// FBs/CSV/FB_EscreveCSVPonteiro
FUNCTION_BLOCK FB_EscreveCSVPonteiro
VAR_INPUT
	bInicia : BOOL;
	sNetId			: T_AmsNetId;	(* TwinCAT system network address *)
	sFileName	: T_MaxString;(* CSV destination file path and name *)
	MAX_CSV_COLUMNS : UINT;
	MAX_CSV_ROWS	: UINT;
	ppDataBase : POINTER TO POINTER TO STRING(255);
END_VAR
VAR_IN_OUT
	//database : ARRAY[*,*] OF STRING(255);
END_VAR
VAR_OUTPUT
	bBusy			: BOOL;
	bError			: BOOL;
	nErrId			: UDINT;
	nRow	 		: UDINT 	:= 0;(* Row number (record) *)
END_VAR
VAR
	bWrite			: BOOL := FALSE;(* Rising edge starts program execution *)
	sCSVLine		: T_MaxString := '';(* Single CSV text line (row, record), we are using string as record buffer (your are able to see created fields) *)
	sCSVField		: T_MaxString := '';(* Single CSV field value (column, record field) *)
	nColumn		: UDINT 	:= 0;(* Column number (record field) *)
	hFile			: UINT		:= 0;(* File handle of the source file *)
	step			: DWORD 	:= 0;
	fbFileOpen	: FB_FileOpen;(* Opens file *)
	fbFileClose	: FB_FileClose;(* Closes file *)
	fbFilePuts		: FB_FilePuts;(* Writes one record (line) *)
	fbWriter		: FB_CSVMemBufferWriter;(* Helper function block used to create CSV data bytes (single record line) *)
	rtInicia		: R_TRIG;
	

	MAX_CSV_FIELD_LENGTH : UDINT := 255;
END_VAR

IF xLicensaValida87208720 THEN
	
//Criado por Tiago Bortolini Cunico
	
	
	CASE step OF
		0:	(* Wait for rising edge at bWrite variable *)
			rtInicia(CLK:=bInicia , Q=> );//gera borda de subina quando liga	
			IF rtInicia.q THEN
				bWrite := TRUE;
			END_IF
			
			IF bWrite THEN
				bWrite 		:= FALSE;
				bBusy 		:= TRUE;
				bError		:= FALSE;
				nErrId		:= 0;
				hFile		:= 0;
				nRow	 	:= 0;
				nColumn		:= 0;
				step 		:= 1;
			END_IF
	
		1:	(* Open source file *)
			fbFileOpen(  bExecute := FALSE  );
			fbFileOpen( 	sNetId := sNetId, sPathName := sFileName, nMode := FOPEN_MODEAPPEND OR FOPEN_MODETEXT,(* Open file in TEXT mode!   FOPEN_MODEWRITE OR FOPEN_MODETEXT*)
							ePath := PATH_GENERIC, bExecute := TRUE );
			step := 2;
	
		2:(* Wait until open not busy *)
			fbFileOpen( bExecute := FALSE, bError => bError, nErrID => nErrID, hFile => hFile );
			IF NOT fbFileOpen.bBusy THEN
				IF NOT fbFileOpen.bError THEN
					step := 3;
				ELSE(* Error: file not found? *)
					step := 100;
				END_IF
			END_IF
	
		3:(* Convert one PLC record to CSV format *)
			sCSVLine := '';
			fbWriter.eCmd := eEnumCmd_First;(* Write first field value *)
			IF nRow < MAX_CSV_ROWS THEN
	
				FOR nColumn := 0 TO MAX_CSV_COLUMNS - 1 BY 1 DO	
					IF  ppDataBase <> 0 AND ppDataBase[nColumn] <> 0 THEN
						IF ppDataBase[nColumn][nRow] <>  '' THEN 
				
							sCSVField := STRING_TO_CSVFIELD( ppDataBase[nColumn][nRow], TRUE );(* TODO: Get field value from your application *)//sCSVField := STRING_TO_CSVFIELD( database[ nRow, nColumn ], FALSE );(* TODO: Get field value from your application *)
							
							(* Add new field to the record buffer *)
							fbWriter( 	pBuffer := ADR( sCSVLine ), cbBuffer := SIZEOF( sCSVLine ) - 1, putValue := sCSVField, pValue := 0, cbValue := 0,
										bCRLF := ( nColumn = MAX_CSV_COLUMNS-1 ) );(* bCRLF == TRUE => Write CRLF after the last field value *)
							IF fbWriter.bOk THEN
								fbWriter.eCmd := eEnumCmd_Next;(* Write next field value *)
							ELSE(* Error *)
								step := 100;
								RETURN;
							END_IF
						END_IF
					ELSE
						step := 100;
					END_IF
				END_FOR(* FOR nColumn := 0... *)
	
				(* FB_FilePuts adds allready CR (carriage return) to the written line.
				We have to replace the $R$L characters with $L character to avoid double CR. *)
				
				IF RIGHT( sCSVLine, 2 ) = '$R$L' THEN //IF RIGHT( sCSVLine, 2 ) = '$R$L' THEN
					sCSVLine := REPLACE( sCSVLine, '$L', 2, LEN( sCSVLine ) - 1 );
				END_IF
				
				nRow := nRow + 1;(* Increment number of created records (rows) *)
				step := 4;(* Write record to the file *)
				
	
			ELSE(* All rows written => Close file *)
				step := 10;
			END_IF
	
		4:	(* Write single text line *)
			fbFilePuts( bExecute := FALSE );
			fbFilePuts( sNetId := sNetId, hFile := hFile, sLine := sCSVLine, bExecute := TRUE );
			step := 5;
	
		5:(* Wait until write not busy *)
			fbFilePuts( bExecute := FALSE, bError => bError, nErrID => nErrID );
			IF NOT fbFilePuts.bBusy THEN
				IF NOT fbFilePuts.bError THEN
					step := 3;(* Write next record *)
				ELSE(* Error *)
					step := 100;
				END_IF
			END_IF
	
		10:	(* Close source file *)
			fbFileClose( bExecute := FALSE );
			fbFileClose( sNetId := sNetId, hFile := hFile, bExecute := TRUE );
			step := 11;
	
		11:(* Wait until close not busy *)
			fbFileClose( bExecute := FALSE, bError => bError, nErrID => nErrID );
			IF ( NOT fbFileClose.bBusy ) THEN
				hFile := 0;
				step := 100;
			END_IF
	
		100: (* Error or ready step => cleanup *)
			IF ( hFile <> 0 ) THEN
				step := 10; (* Close the source file *)
			ELSE
				bBusy := FALSE;
				step := 0;	(* Ready *)
			END_IF
	
	END_CASE

ELSE
	ValidaLicensa();
END_IF

END_FUNCTION_BLOCK

// FBs/Diagnostico/CAN/fb_Diag_CAN
FUNCTION_BLOCK fb_Diag_CAN
VAR_IN_OUT
	stCanDiag : st_Diag_CAN;
END_VAR
VAR_OUTPUT
END_VAR
VAR
	i : INT;
	j : INT := 1;
	
END_VAR

IF xLicensaValida87208720 THEN
	

	stCanDiag.xBusOFF			:= (2#0000_0000_0000_0001 AND stCanDiag.uCanState) > 0;
	stCanDiag.xCanWarning		:= (2#0000_0000_0000_0010 AND stCanDiag.uCanState) > 0;
	stCanDiag.xRxOverrun		:= (2#0000_0000_0000_0100 AND stCanDiag.uCanState) > 0;
	stCanDiag.xCANSendError		:= (2#0000_0000_0001_0000 AND stCanDiag.uCanState) > 0;
	stCanDiag.xFilaRxOverflow	:= (2#0000_0000_0100_0000 AND stCanDiag.uCanState) > 0;
	stCanDiag.xFilaTxOverflow	:= (2#0000_0000_1000_0000 AND stCanDiag.uCanState) > 0;
	
	FOR i := 1 TO 126 DO
	
		IF stCanDiag.uNodeState[i] = 0 THEN
			stCanDiag.xNoOk[i]		:= TRUE;
			stCanDiag.sEstadoNo[i]	:= 'OK';
			CONTINUE;
		END_IF
	
		CASE stCanDiag.uNodeState[i] OF
			1:
				stCanDiag.xNoOk[i]		:= FALSE;
				stCanDiag.sEstadoNo[i]	:= 'Node deactivated';
				CONTINUE;
	
			2:
				stCanDiag.xNoOk[i]		:= FALSE;
				stCanDiag.sEstadoNo[i]	:= 'Node not found';
				CONTINUE;
	
			4:
				stCanDiag.xNoOk[i]		:= FALSE;
				stCanDiag.sEstadoNo[i]	:= 'SDO syntax error at StartUp';
				CONTINUE;
	
			5:
				stCanDiag.xNoOk[i]		:= FALSE;
				stCanDiag.sEstadoNo[i]	:= 'SDO data mismatch at StartUp';
				CONTINUE;
	
			8:
				stCanDiag.xNoOk[i]		:= TRUE;
				stCanDiag.sEstadoNo[i]	:= 'Node StartUp in progress';
				CONTINUE;
	
			11:
				stCanDiag.xNoOk[i]		:= FALSE;
				stCanDiag.sEstadoNo[i]	:= 'CAN-Controller is Bus-OFF';
				CONTINUE;
	
			12:
				stCanDiag.xNoOk[i]		:= TRUE;
				stCanDiag.sEstadoNo[i]	:= 'Pre-Operational';
				CONTINUE;
	
			13:
				stCanDiag.xNoOk[i]		:= FALSE;
				stCanDiag.sEstadoNo[i]	:= 'Server bus fault';
				CONTINUE;
	
			14:
				stCanDiag.xNoOk[i]		:= FALSE;
				stCanDiag.sEstadoNo[i]	:= 'Guarding: toggle error';
				CONTINUE;
	
			20:
				stCanDiag.xNoOk[i]		:= FALSE;
				stCanDiag.sEstadoNo[i]	:= 'TxPDO too short';
				CONTINUE;
	
			22:
				stCanDiag.xNoOk[i]		:= FALSE;
				stCanDiag.sEstadoNo[i]	:= 'Expected TxPDO is missing';
				CONTINUE;
	
			23:
				stCanDiag.xNoOk[i]		:= TRUE;
				stCanDiag.sEstadoNo[i]	:= 'Node is Operational but not all TxPDOs were received';
				CONTINUE;
	
			31:
				stCanDiag.xNoOk[i]		:= TRUE;
				stCanDiag.sEstadoNo[i]	:= 'only for EtherCAT gateways: WC-State of cyclic EtherCAT frame is 1';
				CONTINUE;
		END_CASE
	
		IF stCanDiag.uNodeState[i] > 63 THEN
			stCanDiag.xNoOk[i]		:= TRUE;
			stCanDiag.sEstadoNo[i]	:= 'startup of slave is finished';
			CONTINUE;
		END_IF
	
	END_FOR
	
	i := j;

END_IF

END_FUNCTION_BLOCK

// FBs/Diagnostico/Ethercat/FB_EtherCATDiag
FUNCTION_BLOCK FB_EtherCATDiag
VAR_IN_OUT
	Diagnostico 				: st_DiagnosticoEthercat;
END_VAR
VAR_INPUT
END_VAR
VAR_OUTPUT
	bEtherCATOK					: BOOL;			// no problem on EtherCAT
	bFrameWcStateError			: BOOL;			// error in at least one frame
	bSlaveCountError			: BOOL;			// EtherCAT slave count mismatch (# of cfg slaves <> # of found slaves)
	bMasterDevStateError		: BOOL;			// error in master device state
	bBarramentoInterrompido 	: BOOL;				// caso o barramento esteja interrompido
	stMasterDevState			: ST_EcMasterDevState; // splitted master device state
	bBusy						: BOOL;			// FB busy
	bError						: BOOL;			// FB with error
	iErrorID					: UDINT;		// FB error ID
END_VAR
VAR
	sMasterNetID				: T_AmsNetId; 	// AmsNetId of the EtherCAT master device 
		
	tTimeout					: TIME := T#5S; // ads timeout
	
	iState						: INT;
	nMasterDevStatePrev			: WORD;
	bSlaveCountErrorPrev		: BOOL;
	bAllFrameWcStatesOKPrev		: BOOL;
	bDiagReq					: BOOL := TRUE;
	I							: UDINT;

	(* -- Get Slave Addresses *)
	fbGetSlaveAddresses 		: FB_EcGetAllSlaveAddr;
	arrSlaveAddresses 			: ARRAY[0..255] OF UINT;
	iNumOfSlavesRead			: UINT;

	(* -- Get Slave States *)
	fbGetAllSlaveStates			: FB_EcGetAllSlaveStates;
	arrSlaveStates 				: ARRAY[0..255] OF ST_EcSlaveState;

	(* -- Get Topology Data *)
	iTopologyData				: UDINT;
	fbGetTopologyData			: ADSREAD;
	arrTopologyData				: ARRAY[0..255] OF ST_TopologyData;

	(* -- Check Topology *)
	iDiagIndex					: ARRAY [0..255] OF UINT;
	iDiagPort					: ARRAY [0..255] OF UINT;
	iIdx						: DINT;

	(* -- Scan Slaves *)
	fbEcGetScannedSlaves		: FB_EcGetScannedSlaves;
	arrScannedSlaveInfo			: ARRAY [0..255] OF ST_EcSlaveScannedData;
	nScannedSlaves				: UINT;

	(* -- Get Slave Identities *)
	fbGetSlaveIdentity			: FB_EcGetSlaveIdentity;
	stIdentity 					: ST_EcSlaveIdentity;

	(* -- Get Slave Names *)
	fbGetSlaveName 				: IOF_GetBoxNameByAddr;
	strName						: STRING;

	arrSlaveInfo 				: ARRAY [0..255] OF ST_SlaveStateInfo;
	arrSlaveInfoScanned			: ARRAY [0..255] OF ST_SlaveStateInfoScanned;
	
	xAtualiza 					: BOOL;		
	iAux : INT;
END_VAR



Diagnostico.sEcMasterNetId := F_CreateAmsNetId(nIds := Diagnostico.arrEcMasterNetId);

Diagnostico.fbEtherCATFrameDiag(
	wFrmXWcState 	:= Diagnostico.wFrmXWcState,
	wReqZeroMask 	:= Diagnostico.wReqZeroMask,
	bFrameWcStateOK	=> Diagnostico.bFrameWcStateOK
);

bFrameWcStateError := NOT Diagnostico.bFrameWcStateOK;

bBarramentoInterrompido := Diagnostico.bBarramentoInterrompido := Diagnostico.nEcMasterSlaveCount <> 0 AND Diagnostico.nEcMasterSlaveCount2 <> 0;

bSlaveCountError := (Diagnostico.nEcMasterSlaveCount + Diagnostico.nEcMasterSlaveCount2 <> Diagnostico.nEcMasterSlaveCountCfg) OR (Diagnostico.nEcMasterSlaveCount + Diagnostico.nEcMasterSlaveCount2 = 0);
IF (bSlaveCountError AND NOT bSlaveCountErrorPrev) OR (NOT bSlaveCountError AND bSlaveCountErrorPrev) THEN
	bSlaveCountErrorPrev := bSlaveCountError;
	bDiagReq := TRUE; // slave count error change detected --> diag required
END_IF

IF (Diagnostico.bFrameWcStateOK AND NOT bAllFrameWcStatesOKPrev) OR (NOT Diagnostico.bFrameWcStateOK AND bAllFrameWcStatesOKPrev) THEN
	bAllFrameWcStatesOKPrev := Diagnostico.bFrameWcStateOK;
	bDiagReq := TRUE; // frame error change detected --> diag required
END_IF

IF (Diagnostico.nEcMasterDevState <> nMasterDevStatePrev) THEN
	M_CheckMasterDevState();
	bDiagReq := TRUE; // devstate change detected --> diag required
END_IF

(* acyclic diag *)

IF xAtualiza THEN
	iState := iAux;
END_IF


CASE iState OF
0: (* IDLE *)
	IF bDiagReq THEN				// diag requested
		bDiagReq := FALSE;

		IF Diagnostico.sEcMasterNetId <> '' AND Diagnostico.sEcMasterNetId <> '0.0.0.0.0.0' THEN
			//iState := 1;	// execute diag
			bBusy := TRUE;
		ELSE
			bError := TRUE;
			iErrorID := 7;
		END_IF

		bEtherCATOK := FALSE;
	ELSE
		// check for changes in idle
		IF (bSlaveCountError OR bMasterDevStateError OR NOT Diagnostico.bFrameWcStateOK) AND NOT (arrSlaveInfo[iDiagIndex[0]].bDiagData) THEN
			bEtherCATOK := FALSE;
			bDiagReq := TRUE;//new error --> diag requested
		ELSIF (bSlaveCountError AND NOT bSlaveCountErrorPrev) OR (NOT bSlaveCountError AND bSlaveCountErrorPrev) THEN
			bSlaveCountErrorPrev := bSlaveCountError;
			bEtherCATOK := FALSE;
			bDiagReq := TRUE;// slave count error change detected --> diag required
		ELSIF (Diagnostico.nEcMasterDevState <> nMasterDevStatePrev) THEN
			bEtherCATOK := FALSE;
			bDiagReq := TRUE;// devstate change detected --> diag required
		ELSIF (Diagnostico.bFrameWcStateOK AND NOT bAllFrameWcStatesOKPrev) OR (NOT Diagnostico.bFrameWcStateOK AND bAllFrameWcStatesOKPrev) THEN
			bAllFrameWcStatesOKPrev := Diagnostico.bFrameWcStateOK;
			bEtherCATOK := FALSE;
			bDiagReq := TRUE;// frame error change detected --> diag required
		ELSIF (bSlaveCountError OR bMasterDevStateError OR NOT Diagnostico.bFrameWcStateOK OR arrSlaveInfo[iDiagIndex[0]].bDiagData) THEN
			bEtherCATOK := FALSE;
		ELSE
			bEtherCATOK := TRUE;
		END_IF
	END_IF
(*
1: (* get adresses *)
	M_GetSlaveAdresses_1();

2: (* get states *)
	M_GetSlaveStates_2();

3:	(* get topology data length *)
	M_GetTopoDataLen_3();

4:	(* get topology data *)
	M_GetTopoData_4();

5:	(* scan slaves *)
	M_ScanSlaves_5();

6:	(* get identity *)
	M_GetSlaveIdentity_6();

7:	(* get name *)
	M_GetSlaveName_7();

8:	(* get scanned name *)
	M_GetScannedSlaveName_8();

10:	(* DONE *)
	bBusy := FALSE;
	iState := 0;
*)

END_CASE

ACTION M_CheckMasterDevState:
(* check master errors based on devstate *)
bMasterDevStateError 				:= Diagnostico.nEcMasterDevState <> 0;
stMasterDevState.bLinkError 		:= ((Diagnostico.nEcMasterDevState AND 16#000F) = 1) OR ((Diagnostico.nEcMasterDevState AND 16#000F) = 4);
stMasterDevState.bResetRequired 	:= ((Diagnostico.nEcMasterDevState AND 16#000F) = 2) OR ((Diagnostico.nEcMasterDevState AND 16#FFF0) = 16#10);
stMasterDevState.bMissFrmRedMode 	:= (Diagnostico.nEcMasterDevState AND 16#000F) = 8;
stMasterDevState.bWatchdogTriggerd 	:= (Diagnostico.nEcMasterDevState AND 16#20) = 16#20;
stMasterDevState.bDriverNotFound 	:= (Diagnostico.nEcMasterDevState AND 16#40) = 16#40;
stMasterDevState.bResetActive 		:= (Diagnostico.nEcMasterDevState AND 16#80) = 16#80;
stMasterDevState.bAtLeastOneNotInOp := ((Diagnostico.nEcMasterDevState AND 16#100) = 16#100) OR ((Diagnostico.nEcMasterDevState AND 16#200) = 16#200) OR
										((Diagnostico.nEcMasterDevState AND 16#400) = 16#400) OR ((Diagnostico.nEcMasterDevState AND 16#800) = 16#800);
stMasterDevState.bDcNotInSync 		:= (Diagnostico.nEcMasterDevState AND 16#1000) = 16#1000;
nMasterDevStatePrev 				:= Diagnostico.nEcMasterDevState;
END_ACTION

ACTION M_GetScannedSlaveName_8:
fbGetSlaveName(
	NETID		:= '',
	DEVICEID	:= Diagnostico.nEcMasterDeviceId,
	BOXADDR		:= arrScannedSlaveInfo[iDiagIndex[iIdx]].nAddr,
	START		:= TRUE,
	TMOUT		:= tTimeout,
	BOXNAME		=> strName
);

IF NOT fbGetSlaveName.BUSY THEN
	fbGetSlaveName(START:= FALSE);

	(* add scanned info *)
	arrSlaveInfoScanned[iDiagIndex[iIdx]].nIndex := iDiagIndex[iIdx] + 1;
	
	IF arrScannedSlaveInfo[iDiagIndex[iIdx]].nAddr <> 0 THEN
		IF NOT fbGetSlaveName.ERR THEN
			arrSlaveInfoScanned[iDiagIndex[iIdx]].sName := strName;
		END_IF
	ELSE
		arrSlaveInfoScanned[iDiagIndex[iIdx]].sType		:= '';
	END_IF

	IF (iDiagIndex[iIdx] < nScannedSlaves) THEN
		arrSlaveInfoScanned[iDiagIndex[iIdx]].sType		:= F_ConvProductCodeToString(arrScannedSlaveInfo[iDiagIndex[iIdx]].stSlaveIdentity);
	ELSE
		arrSlaveInfoScanned[iDiagIndex[iIdx]].sType		:= '';
	END_IF

	arrSlaveInfoScanned[iDiagIndex[iIdx]].nECAddr	:= arrScannedSlaveInfo[iDiagIndex[iIdx]].nAddr;
(* // desativado por agora pra ter uma versao que ja funciona em alguem nivel
	IF arrSlaveInfoScanned[iDiagIndex[iIdx]].sName <> arrSlaveInfo[iDiagIndex[iIdx]].sName THEN
		arrSlaveInfoScanned[iDiagIndex[iIdx]].bDifferentName := TRUE;
	ELSE
		arrSlaveInfoScanned[iDiagIndex[iIdx]].bDifferentName := FALSE;
	END_IF

	IF arrSlaveInfoScanned[iDiagIndex[iIdx]].nECAddr <> arrSlaveInfo[iDiagIndex[iIdx]].nECAddr THEN
		arrSlaveInfoScanned[iDiagIndex[iIdx]].bDifferentAddr := TRUE;
	ELSE
		arrSlaveInfoScanned[iDiagIndex[iIdx]].bDifferentAddr := FALSE;
	END_IF

	IF arrSlaveInfoScanned[iDiagIndex[iIdx]].sType <> arrSlaveInfo[iDiagIndex[iIdx]].sType THEN
		arrSlaveInfoScanned[iDiagIndex[iIdx]].bDifferentType := TRUE;
	ELSE
		arrSlaveInfoScanned[iDiagIndex[iIdx]].bDifferentType := FALSE;
	END_IF
*)	
	//Tiago
	//Joga no arrSlaveInfo o nome/modelo
	(*
	arrSlaveInfo[iDiagIndex[iIdx]].sName := arrSlaveInfoScanned[iDiagIndex[iIdx]].sName;
	arrSlaveInfo[iDiagIndex[iIdx]].nECAddr := arrSlaveInfoScanned[iDiagIndex[iIdx]].nECAddr;
	arrSlaveInfo[iDiagIndex[iIdx]].sType := arrSlaveInfoScanned[iDiagIndex[iIdx]].sType;
	arrSlaveInfo[iDiagIndex[iIdx]].nIndex := arrSlaveInfoScanned[iDiagIndex[iIdx]].nIndex;
	*)
	
	IF iIdx < 255 THEN
		iIdx := iIdx + 1;
		iState := 6;
	ELSE
		iIdx := 0;
		iState := 10;

		FOR I := 0 TO 255 DO
			IF iDiagPort[I] <> 0 THEN
				Diagnostico.arrDiagSlaveInfo[I] := arrSlaveInfo[iDiagIndex[I]];
				Diagnostico.arrDiagSlaveInfoScanned[I] := arrSlaveInfoScanned[iDiagIndex[I]];
			ELSE
				MEMSET(ADR(Diagnostico.arrDiagSlaveInfo[I]), 0, SIZEOF(Diagnostico.arrDiagSlaveInfo[I]));
				MEMSET(ADR(Diagnostico.arrDiagSlaveInfoScanned[I]), 0, SIZEOF(Diagnostico.arrDiagSlaveInfoScanned[I]));
			END_IF
		END_FOR
	END_IF
END_IF
END_ACTION

ACTION M_GetSlaveAdresses_1:
fbGetSlaveAddresses(
	sNetId		:= Diagnostico.sEcMasterNetId,
	pAddrBuf	:= ADR(arrSlaveAddresses),
	cbBufLen	:= SIZEOF(arrSlaveAddresses),
	bExecute	:= TRUE,
	tTimeout	:= tTimeout,
	nSlaves		=> iNumOfSlavesRead
);

IF NOT fbGetSlaveAddresses.bBusy THEN
	fbGetSlaveAddresses(bExecute:= FALSE);
	IF NOT fbGetSlaveAddresses.bError THEN
		FOR I := 0 TO MIN(iNumOfSlavesRead, 255) DO
			arrSlaveInfo[I].nECAddr := arrSlaveAddresses[I];
		END_FOR
	END_IF
	iState := 2;
END_IF
END_ACTION

ACTION M_GetSlaveIdentity_6:
fbGetSlaveIdentity(
	sNetId		:= Diagnostico.sEcMasterNetId,
	nSlaveAddr	:= arrSlaveInfo[iDiagIndex[iIdx]].nECAddr,
	bExecute	:= TRUE,
	tTimeout	:= tTimeout,
	identity	=> stIdentity
);

IF NOT fbGetSlaveIdentity.bBusy THEN
	fbGetSlaveIdentity(bExecute:= FALSE);

	IF NOT fbGetSlaveIdentity.bError THEN
			arrSlaveInfo[iDiagIndex[iIdx]].nIndex	:= iDiagIndex[iIdx] + 1;
			arrSlaveInfo[iDiagIndex[iIdx]].sType 	:= F_ConvProductCodeToString(stSlaveIdentity := stIdentity);
	END_IF
	iState := 7;
END_IF
END_ACTION

ACTION M_GetSlaveName_7:
fbGetSlaveName(
	NETID		:= '',
	DEVICEID	:= Diagnostico.nEcMasterDeviceId,
	BOXADDR		:= arrSlaveInfo[iDiagIndex[iIdx]].nECAddr,
	START		:= TRUE,
	TMOUT		:= tTimeout,
	BOXNAME		=> strName
);

IF NOT fbGetSlaveName.BUSY THEN
	fbGetSlaveName(START:= FALSE);

	IF NOT fbGetSlaveName.ERR THEN
			arrSlaveInfo[iDiagIndex[iIdx]].sName 	:= strName;
	END_IF

	iState := 8;
END_IF
END_ACTION

ACTION M_GetSlaveStates_2:
fbGetAllSlaveStates(
	sNetId		:= Diagnostico.sEcMasterNetId,
	pStateBuf	:= ADR(arrSlaveStates),
	cbBufLen	:= SIZEOF(arrSlaveStates),
	bExecute	:= TRUE,
	tTimeout	:= tTimeout,
	nSlaves		=> iNumOfSlavesRead
);

IF NOT fbGetAllSlaveStates.bBusy AND fbGetAllSlaveStates.bExecute THEN
	fbGetAllSlaveStates(bExecute:= FALSE);

	IF NOT fbGetAllSlaveStates.bError THEN
		IF iNumOfSlavesRead = Diagnostico.nEcMasterSlaveCountCfg THEN
			FOR I := 0 TO 255 DO
				iDiagIndex[I] := 0;
			END_FOR

			(* split slave state and link state *)
			FOR I := 0 TO MIN(iNumOfSlavesRead, 255) DO	
				(* slave state*)
				arrSlaveInfo[I].stState.eEcState 		:= arrSlaveStates[I].deviceState AND 16#0F;
				arrSlaveInfo[I].stState.bError 			:= arrSlaveStates[I].deviceState.4;
				arrSlaveInfo[I].stState.bInvalidVPRS 	:= arrSlaveStates[I].deviceState.5;
				(* link state *)
				arrSlaveInfo[I].stState.bNoCommToSlave 	:= arrSlaveStates[I].linkState.0;
				arrSlaveInfo[I].stState.bLinkError 		:= arrSlaveStates[I].linkState.1;
				arrSlaveInfo[I].stState.bMissingLink 	:= arrSlaveStates[I].linkState.2;
				arrSlaveInfo[I].stState.bUnexpectedLink := arrSlaveStates[I].linkState.3;
				arrSlaveInfo[I].stState.bPortA 			:= arrSlaveStates[I].linkState.4;
				arrSlaveInfo[I].stState.bPortB 			:= arrSlaveStates[I].linkState.5;
				arrSlaveInfo[I].stState.bPortC 			:= arrSlaveStates[I].linkState.6;
				arrSlaveInfo[I].stState.bPortD 			:= arrSlaveStates[I].linkState.7;
				(* DiagData *)
				arrSlaveInfo[I].bDiagData	:= ((arrSlaveStates[I].deviceState AND 16#F0) <> 0) OR
					(((arrSlaveStates[I].deviceState AND 16#0F) > 0) AND ((arrSlaveStates[I].deviceState AND 16#0F) < 8)) OR
					(arrSlaveStates[I].linkState <> 0);

				IF arrSlaveInfo[I].bDiagData THEN
					IF (I=0) THEN
						iDiagIndex[0] := 0;
					ELSE
						IF (iDiagIndex[0] = 0) AND NOT arrSlaveInfo[0].bDiagData THEN
							iDiagIndex[0] :=  UDINT_TO_UINT(I);
						END_IF
					END_IF
				END_IF
			END_FOR
		END_IF
	END_IF

	iState := 3;

 // nao entendi oq ele ta fazendo aqui, vou tirar por agora
 (*
	IF arrSlaveInfo[iDiagIndex[0]].bDiagData THEN
		iState := 3;
	ELSE
		FOR I := 0 TO 255 DO
			MEMSET(ADR(Diagnostico.arrDiagSlaveInfo[I]), 0, SIZEOF(Diagnostico.arrDiagSlaveInfo[I]));
			MEMSET(ADR(Diagnostico.arrDiagSlaveInfoScanned[I]), 0, SIZEOF(Diagnostico.arrDiagSlaveInfoScanned[I]));
		END_FOR
		iState := 3;
		//iState := 10;
	END_IF
*)
END_IF
END_ACTION

ACTION M_GetTopoData_4:
fbGetTopologyData(
	NETID	:= Diagnostico.sEcMasterNetId,
	PORT	:= 16#FFFF,
	IDXGRP	:= 16#22,
	IDXOFFS	:= 0,
	LEN		:= iTopologyData*SIZEOF(arrTopologyData[0]),
	DESTADDR:= ADR(arrTopologyData),
	READ	:= TRUE,
	TMOUT	:= tTimeout,
);


IF NOT fbGetTopologyData.BUSY THEN
	fbGetTopologyData(READ := FALSE);

	
	IF NOT fbGetTopologyData.ERR THEN

	
		FOR I := 0 TO iTopologyData-1 DO
			iDiagIndex[i] := arrTopologyData[i].iOwnPhysicalAddr-1000;
			
		END_FOR
	
	
	 // a logica que ta aqui na real é feita assim pq no exemplo o cara usa um barramento que tem so 4 cartao ai logo na primeira ele consegue
	 // ler todos os enderessos, so que o jamelao nao fez o esquema que desse pra ler todos de qualquer barramento
		
(*
		(* clear diag index  *)
		FOR I := 0 TO 255 DO
			iDiagIndex[i] := 0;
		END_FOR
	

		FOR I := 0 TO 10 DO
			
			iDiagPort[0] := arrTopologyData[iDiagIndex[i]].iOwnPhysicalAddr;
			iDiagPort[1] := arrTopologyData[iDiagIndex[i]].stPhysicalAddr.portB;
			iDiagPort[2] := arrTopologyData[iDiagIndex[i]].stPhysicalAddr.portC;
			iDiagPort[3] := arrTopologyData[iDiagIndex[i]].stPhysicalAddr.portD;
		
			(* find slaves on PortB of first slave with diag *)
			IF iDiagPort[i] <> 0 THEN
				FOR I := 0 TO MIN(iTopologyData-1,255) DO
					IF arrTopologyData[I].iOwnPhysicalAddr = iDiagPort[i] THEN
						iDiagIndex[1] := UDINT_TO_UINT(I);
						EXIT;
					END_IF
				END_FOR
			END_IF
	
			(* find slaves on PortC of first slave with diag *)
			IF iDiagPort[i] <> 0 THEN
				FOR I := 0 TO MIN(iTopologyData-1,255) DO
					IF arrTopologyData[I].iOwnPhysicalAddr = iDiagPort[i] THEN
						iDiagIndex[2] := UDINT_TO_UINT(I);
						EXIT;
					END_IF
				END_FOR
			END_IF
	
			(* find slaves on PortD of first slave with diag *)
			IF iDiagPort[i] <> 0 THEN
				FOR I := 0 TO MIN(iTopologyData-1,255) DO
					IF arrTopologyData[I].iOwnPhysicalAddr = iDiagPort[i] THEN
						iDiagIndex[3] := UDINT_TO_UINT(I);
						EXIT;
					END_IF
				END_FOR
			END_IF
		END_FOR
*)
	END_IF
	

	iIdx := 0;
	iState := 5;
END_IF
END_ACTION

ACTION M_GetTopoDataLen_3:
fbGetTopologyData(
	NETID	:= Diagnostico.sEcMasterNetId,
	PORT	:= 16#FFFF,
	IDXGRP	:= EC_ADS_IGRP_MASTER_COUNT_SLAVE,
	IDXOFFS	:= EC_ADS_IOFFS_MASTER_COUNT_SLAVE,
	LEN		:= SIZEOF(iTopologyData),
	DESTADDR:= ADR(iTopologyData),
	READ	:= TRUE,
	TMOUT	:= tTimeout,
);

IF NOT fbGetTopologyData.BUSY THEN
	fbGetTopologyData(READ := FALSE);

	iState := 4;
END_IF
END_ACTION

ACTION M_ScanSlaves_5:
fbEcGetScannedSlaves(
	bExecute				:= TRUE,
	sNetId					:= Diagnostico.sEcMasterNetId,
	pArrEcScannedSlaveInfo	:= ADR(arrScannedSlaveInfo),
	cbBufLen				:= SIZEOF(arrScannedSlaveInfo),
	tTimeout				:= tTimeout
);

IF NOT fbEcGetScannedSlaves.bBusy THEN
	fbEcGetScannedSlaves(bExecute := FALSE);
	iState := 6;

	IF fbEcGetScannedSlaves.bError THEN
		nScannedSlaves := 0;
	ELSE
		nScannedSlaves := fbEcGetScannedSlaves.nSlaves;
	END_IF
END_IF
END_ACTION

END_FUNCTION_BLOCK

// FBs/Diagnostico/Ethercat/FB_EtherCATFrameDiag
FUNCTION_BLOCK FB_EtherCATFrameDiag
VAR_INPUT
	wFrmXWcState 		: WORD;				// FrmXWcState
	wReqZeroMask 		: WORD := 16#FFFF;	// mask, bit TRUE: require wFrmXWcState.bit = FALSE, bit FALSE: ignore wFrmXWcState.bit *)
END_VAR
VAR_OUTPUT
	bFrameWcStateOK		: BOOL;				// result of fram state check
END_VAR
VAR
END_VAR

(* mask out ignored error bits and compare result against 0 *)
bFrameWcStateOK := ((wFrmXWcState AND wReqZeroMask) = 0);

END_FUNCTION_BLOCK

// FBs/Diagnostico/Ethernet_PCgeral/FB_Diag_Geral
FUNCTION_BLOCK FB_Diag_Geral
VAR_IN_OUT
	stGeral : st_Diag_PC_Geral;
END_VAR
VAR_OUTPUT
END_VAR
VAR
	
	uiUsoCpu 	: UINT;
	iTempCpu 	: INT;
	uliMemoriaRamUsada	: ULINT;
	rAux : REAL;
	rMemoriaRamUsada : REAL;
	uliespacoLivreHD	: ULINT;
	rEspacoLivreHD : REAL;
	
	xDHCP			: ARRAY[1..20] OF BOOL;
	sIPV4			: ARRAY[1..20] OF STRING(39);
	sIPV4Mask		: ARRAY[1..20] OF STRING;
	sIPV4Nome		: ARRAY[1..20] OF STRING(79);
	sIPV4NomeVirtual: ARRAY[1..20] OF STRING(79);
	NumeroDePortas	: USINT;
	
	sNomeCPU : STRING;
	
	tcVersion : STRING;
	tcAMSNetID : STRING;
	tcSystemID : STRING;
	
	
	
	
	
	hrGetValue		: HRESULT;	
	
	fbDiagnostico		: ARRAY[1..14] OF FB_IPCDiag_ReadParameterPeriodic := [	(eParameterKey:=E_IPCDiag_ParameterKey.CPU_Usage, tPeriod:= T#10S, sNetId:=''),
																		 		(eParameterKey:=E_IPCDiag_ParameterKey.CPU_Temp, tPeriod:= T#10S, sNetId:=''),
																		 		(eParameterKey:=E_IPCDiag_ParameterKey.Memory_ProgramMemoryAllocated, tPeriod:= T#10S, sNetId:=''),
																		 		(eParameterKey:=E_IPCDiag_ParameterKey.Disk_FreeSpaceOfVolumeC, tPeriod:= T#10S, sNetId:=''),
																		 		(eParameterKey:=E_IPCDiag_ParameterKey.NIC_DHCP, tPeriod:= T#10S, sNetId:=''),
																		 		(eParameterKey:=E_IPCDiag_ParameterKey.NIC_IPv4Address, tPeriod:= T#10S, sNetId:=''),
																		 		(eParameterKey:=E_IPCDiag_ParameterKey.NIC_IPv4SubnetMask, tPeriod:= T#10S, sNetId:=''),
																		 		(eParameterKey:=E_IPCDiag_ParameterKey.NIC_ModuleCnt, tPeriod:= T#10S, sNetId:=''),
																		 		(eParameterKey:=E_IPCDiag_ParameterKey.NIC_Name, tPeriod:= T#10S, sNetId:=''),
																		 		(eParameterKey:=E_IPCDiag_ParameterKey.NIC_VirtualDeviceName, tPeriod:= T#10S, sNetId:=''),
																		 		(eParameterKey:=E_IPCDiag_ParameterKey.IPCDeviceName, tPeriod:= T#10S, sNetId:=''),
																		 		(eParameterKey:=E_IPCDiag_ParameterKey.TC_Version, tPeriod:= T#10S, sNetId:=''),
																		 		(eParameterKey:=E_IPCDiag_ParameterKey.TC_AmsNetID, tPeriod:= T#10S, sNetId:=''),
																		 		(eParameterKey:=E_IPCDiag_ParameterKey.TC_SystemID, tPeriod:= T#10S, sNetId:='')];
	

	
	fbDiagRegister		: ARRAY[1..14] OF FB_IPCDiag_Register;
	
	i : INT;


END_VAR

IF xLicensaValida87208720 THEN
	
	
	FOR i:= 1 TO 14 DO
		fbDiagRegister[i](bExecute:= TRUE);
		fbDiagnostico[i](
		bEnable:= TRUE,
		tPeriod:= T#10S, 
		fbRegister:= fbDiagRegister[i]);
	END_FOR
	
	fbDiagnostico[1].GetParameter(pBuffer:=ADR(uiUsoCpu), nBufferSize:=SIZEOF(uiUsoCpu));
	fbDiagnostico[2].GetParameter(pBuffer:=ADR(iTempCpu), nBufferSize:=SIZEOF(iTempCpu));
	fbDiagnostico[3].GetParameter(pBuffer:=ADR(uliMemoriaRamUsada), nBufferSize:=SIZEOF(uliMemoriaRamUsada));
	rAux := ULINT_TO_REAL(uliMemoriaRamUsada);
	rMemoriaRamUsada := rAux/1000000000;
	fbDiagnostico[4].GetParameter(pBuffer:=ADR(uliespacoLivreHD), nBufferSize:=SIZEOF(uliespacoLivreHD));
	rAux := ULINT_TO_REAL(uliespacoLivreHD);
	respacoLivreHD := rAux/1000000000;
	fbDiagnostico[5].GetParameter(pBuffer:=ADR(xDHCP), nBufferSize:=SIZEOF(xDHCP));
	fbDiagnostico[6].GetParameterStrings(pBuffer:=ADR(sIPV4), nBufferSize:=SIZEOF(sIPV4), nStrings:=20);
	fbDiagnostico[7].GetParameterStrings(pBuffer:=ADR(sIPV4Mask), nBufferSize:=SIZEOF(sIPV4Mask), nStrings:=20);
	fbDiagnostico[8].GetParameter(pBuffer:=ADR(NumeroDePortas), nBufferSize:=SIZEOF(NumeroDePortas));
	
	
	hrGetValue := fbDiagnostico[9].GetParameterByIdx(pBuffer:=ADR(sIPV4Nome[1]), nBufferSize:=SIZEOF(sIPV4Nome[1]), 1);
	FOR i:= 2  TO 20 DO
		IF SUCCEEDED(hrGetValue) THEN
			hrGetValue := fbDiagnostico[9].GetParameterByIdx(pBuffer:=ADR(sIPV4Nome[i]), nBufferSize:=SIZEOF(sIPV4Nome[i]), int_to_usint(i));
		END_IF
	END_FOR
	
	
	fbDiagnostico[10].GetParameterStrings(pBuffer:=ADR(sIPV4NomeVirtual), nBufferSize:=SIZEOF(sIPV4NomeVirtual), nStrings:=20);
	
	fbDiagnostico[11].GetParameter(pBuffer:=ADR(sNomeCPU), nBufferSize:=SIZEOF(sNomeCPU));
	fbDiagnostico[12].GetParameter(pBuffer:=ADR(tcVersion), nBufferSize:=SIZEOF(tcVersion));
	fbDiagnostico[13].GetParameter(pBuffer:=ADR(tcAMSNetID), nBufferSize:=SIZEOF(tcAMSNetID));
	fbDiagnostico[14].GetParameter(pBuffer:=ADR(tcSystemID), nBufferSize:=SIZEOF(tcSystemID));
	
	
	
	
	stGeral.NumeroDePortasRede := NumeroDePortas;
	
	FOR i:= 1 TO NumeroDePortas DO
		stGeral.stEthernet[i].sNome := sIPV4NomeVirtual[i];
		stGeral.stEthernet[i].sNomeAdaptador := sIPV4Nome[i];
		stGeral.stEthernet[i].sIP := sIPV4[i];
		stGeral.stEthernet[i].sMask := sIPV4Mask[i];
		stGeral.stEthernet[i].xDHCP := xDHCP[i];
	END_FOR
	
	
	stGeral.uiUsoCpu := uiUsoCpu;
	stGeral.iTempCpu := iTempCpu;
	stGeral.rMemoriaRamUsada := rMemoriaRamUsada;
	stGeral.rEspacoLivreHD := rEspacoLivreHD;
	stGeral.sNomeCPU := sNomeCPU;
	
	stGeral.tcVersion := tcVersion;
	stGeral.tcAMSNetID := tcAMSNetID;
	stGeral.tcSystemID := tcSystemID;


END_IF

END_FUNCTION_BLOCK

// FBs/Geral/FB_FFT
FUNCTION_BLOCK FB_FFT
VAR_INPUT
	xRodaCalculo : BOOL := FALSE; //Sinal Para Rodar Cálculo da FFT
END_VAR

VAR_INPUT RETAIN
	uiLenght	: UINT; 	//Comprimento da Amostragem (256, 512, 1024 ou outro exponencial de base 2)
END_VAR

VAR_OUTPUT
	xFinalizouCalculo	: BOOL := FALSE; //Indica que o Cálculo Finalizou com Sucesso
END_VAR

VAR_IN_OUT
	x_real	: ARRAY [0..511] OF REAL; //Vetor com a componente Real;
	x_complex	: ARRAY[0..511] OF REAL; //Vetor com a componente Imaginária
END_VAR

VAR
	tmp_real		: ARRAY[0..511] OF REAL; //Temporary Storage for real components
	tmp_complex	: ARRAY[0..511] OF REAL; //Temporary Storage for Imaginary Components
	w_real			: ARRAY[0..511] OF REAL;	 //Twiddle factors' real components
	w_complex		: ARRAY[0..511] OF REAL;	 //Twiddle factors' imaginary components
END_VAR

VAR RETAIN
	N				: UINT;		 //Lenght of computed FFT vector	
	k				: UINT;		 //Loop Index
	ind				: UINT;		 //Index of first even sum element
	w_ind			: UINT;		 //Twiddle factor index
	span			: UINT;		 //Block index
	LpN				: UINT;		 //Total Data lenght divided by current N, Saved for optimization reasons
	w_r				: REAL;		 //Selected twiddle factor real component
	w_c				: REAL;		 //Selected twiddle factor imaginary component
	A_r				: REAL;		 //Even Element real component
	A_c				: REAL;		 //Even Element imaginary component
	B_r				: REAL;		 //Odd Element real component
	B_c				: REAL;		 //Odd Element imaginary component
END_VAR



IF xLicensaValida87208720 THEN
		
	
	IF xRodaCalculo THEN
		N := 2;
		WHILE N <= uiLenght DO
				(* Twidddle factor precalculation *)
				FOR k := 0 TO N/8 DO
					w_real[k] := COS(2.0*3.14159265359*UINT_TO_REAL(k)/UINT_TO_REAL(N));
					w_complex[k] := SIN(2.0*3.14159265359*UINT_TO_REAL(k)/UINT_TO_REAL(N));
				END_FOR;
				
				ind := 0;
				w_ind := 0;
				span := 1;
				LpN := uiLenght/N;
				FOR k := 0 TO uiLenght-1 DO
					
					(* Selecting right twiddle factor
					   Cases are split in two just to halve condition evaluations *)
					IF w_ind <= N/2 THEN
						IF w_ind <= N/8 THEN					
							w_r := w_real[ w_ind ];
							w_c := -w_complex[ w_ind ];
						ELSIF w_ind <= N/4 THEN					
							w_r := w_complex[ N/4-w_ind ];
							w_c := -w_real[ N/4-w_ind ];
						ELSIF w_ind <= 3*N/8 THEN					
							w_r := -w_complex[ w_ind-N/4 ];
							w_c := -w_real[ w_ind-N/4 ];
						ELSE					
							w_r := -w_real[ N/2-w_ind ];
							w_c := -w_complex[ N/2-w_ind ];
						END_IF;
					ELSE
						IF w_ind <= 5*N/8 THEN
							w_r := -w_real[ w_ind-N/2 ];
							w_c := w_complex[ w_ind-N/2 ];
						ELSIF w_ind <= 3*N/4 THEN
							w_r := -w_complex[ 3*N/4-w_ind ];
							w_c := w_real[ 3*N/4-w_ind ];
						ELSIF w_ind <= 7*N/8 THEN
							w_r := w_complex[ w_ind-3*N/4 ];
							w_c := w_real[ w_ind-3*N/4 ];
						ELSE
							w_r := w_real[ N-w_ind ];
							w_c := w_complex[ N-w_ind ];
						END_IF;
					END_IF;
		   
					(* Summation of two elements, with odd element multipication with twiddle
					   A + B*w = (A_r+iA_c)+(B_r+iB_c)(W_r+iW_c)
					*)
					A_r := x_real[ ind ];
					A_c := x_complex[ ind ];
					B_r := x_real[ ind+LpN ];
					B_c := x_complex[ ind+LpN ];
					
					(* Separation of real and imaginary components *)
					tmp_real[ k ] := A_r + B_r*w_r - B_c*w_c;
					tmp_complex[ k ] := A_c + B_r*w_c + B_c*w_r;
					
					(* Indexing
					   Index is the index of even element. Odd element is always with index
					   offset of LpN from even element. *)
					ind := ind + 1;
					IF ind + LpN = uiLenght THEN (* Transition from first half to second *)
						ind := 0;
						w_ind := w_ind + 1;
						span  := 1;
					ELSIF ind + LpN = span*LpN*2 THEN (* Transition between spans *)
						ind := ind + LpN;
						w_ind := w_ind + 1;
						span := span + 1;
					END_IF;
		
				END_FOR;
				N := N*2;
				
				(* Copy all elements from temp to data vector *)
				FOR k := 0 TO uiLenght-1 DO
					x_real[k] := tmp_real[k];
					x_complex[k] := tmp_complex[k];
				END_FOR;	
		END_WHILE;
	
		xFinalizouCalculo:=TRUE;
	ELSE
		xFinalizouCalculo:=FALSE;	
	END_IF

ELSE
	ValidaLicensa();
END_IF

END_FUNCTION_BLOCK

// FBs/Geral/FB_HorimetroTime_Preciso
FUNCTION_BLOCK FB_HorimetroTime_Preciso
VAR_INPUT
	xConta : BOOL;
	xReset : BOOL;
END_VAR
VAR_OUTPUT
	Tempo : TIME;
END_VAR
VAR
	systime         		: GETSYSTEMTIME;
	currentTime     		: T_FILETIME;
	dwlowAnterior 			: DWORD;
	rtReset : R_TRIG;


END_VAR


IF xLicensaValida87208720 THEN
	
	
	systime(timeLoDw => currentTime.dwLowDateTime, timeHiDW => currentTime.dwHighDateTime);
	
	rtReset(CLK:= xReset, Q=> );
	
	IF rtReset.q THEN
		Tempo := T#0S;
	END_IF
	
	
	IF (dwlowAnterior <> (currentTime.dwLowDateTime/10000000)) AND xConta THEN
		
		Tempo := Tempo + T#1S;
	END_IF
	
	dwlowAnterior := currentTime.dwLowDateTime/10000000;


ELSE
	ValidaLicensa();
END_IF

END_FUNCTION_BLOCK

// FBs/Geral/FB_RodaTextoString
FUNCTION_BLOCK FB_RodaTextoString
VAR_INPUT
	tParadoInicio : TIME := T#5S;
	tParadoFinal : TIME := T#5S;
	tTrocaLetra : TIME := T#1S;
	sStringTotal : STRING;
	iTamanhoStringSaida : INT := 10;
END_VAR
VAR_OUTPUT
	sStringRodando : STRING;
END_VAR
VAR
	tonRodando : TON;
	iEstado : INT;
	iQuantosApagar : INT;
	iQuantosCaracters : INT;
END_VAR


iQuantosCaracters := LEN(sStringTotal);


CASE iEstado OF
	
	0:// conta o tempo de inicio 
		sStringRodando := LEFT(sStringTotal,iTamanhoStringSaida);
		tonRodando(IN:= TRUE, PT:= tParadoInicio, Q=> , ET=> );
		IF tonRodando.q THEN
			tonRodando(IN:= FALSE);
			iEstado := 1;
			iQuantosApagar := 0;
		END_IF
		
	1://conta o tempo e vai rodando
	
		tonRodando(IN:= TRUE, PT:= tTrocaLetra, Q=> , ET=> );
		IF tonRodando.q THEN
			tonRodando(IN:= FALSE);
			iEstado := 1;
			iQuantosApagar := iQuantosApagar + 1;
		END_IF
		
		sStringRodando := DELETE(sStringTotal,iQuantosApagar,0);
		sStringRodando := LEFT(sStringRodando,iTamanhoStringSaida);
		
		IF iTamanhoStringSaida + iQuantosApagar > iQuantosCaracters THEN
			tonRodando(IN:= FALSE);
			iEstado := 2;
		END_IF
	
	2:// conta o tempo do fim 
	
		sStringRodando := DELETE(sStringTotal,iQuantosApagar,0);
		
		tonRodando(IN:= TRUE, PT:= tParadoFinal, Q=> , ET=> );
		IF tonRodando.q THEN
			tonRodando(IN:= FALSE);
			iEstado := 0;
		END_IF
		
END_CASE

END_FUNCTION_BLOCK

// FBs/Graficos/GraficoTF2000/FB_GraficoTF2000
FUNCTION_BLOCK FB_GraficoTF2000
VAR_INPUT
	Valor : REAL;
	TempoEntreCadaAmostra : TIME;
	emXColocarTimespamp : BOOL := TRUE;
END_VAR
VAR_IN_OUT
	Vetor : ARRAY[*] OF ST_Grafico;
END_VAR
VAR_OUTPUT
END_VAR
VAR
	
	fb_HoraAgora : FB_LocalSystemTime;
	tsAgora : TIMESTRUCT;

	iMinVetor : DINT := -1;
	iMaxVetor : DINT := -1;
	
	iControle : DINT;
	
	tonControle : TON;

	ANYtype_TO_REAL: INT;
	
	I : DINT;

	sAux : ARRAY[1..5] OF STRING(255);
	sAux2 : STRING;
	
	xMudou : BOOL;
END_VAR


IF xLicensaValida87208720 THEN
		
	
	//Criado por Tiago Bortolini Cunico
	
	IF emXColocarTimespamp THEN
		fb_HoraAgora(
			sNetID:='' , 
			bEnable:=TRUE , 
			dwCycle:= , 
			dwOpt:= , 
			tTimeout:= , 
			bValid=> , 
			systemTime=> tsAgora, 
			tzID=> );
	END_IF
	
	IF (iMinVetor <> LOWER_BOUND(Vetor,1) OR iMaxVetor <> UPPER_BOUND(Vetor,1)) THEN
		xMudou := TRUE;
		iMinVetor := LOWER_BOUND(Vetor,1);
		iMaxVetor := UPPER_BOUND(Vetor,1);
	END_IF
	
	
	IF xMudou AND (fb_HoraAgora.bValid AND emXColocarTimespamp) THEN
		
		IF tsAgora.wHour < 10 THEN
			sAux[1] := CONCAT('0',WORD_TO_STRING(tsAgora.wHour));
		ELSE
			sAux[1] := WORD_TO_STRING(tsAgora.wHour);
		END_IF
		sAux[2] := ':';
		
		IF tsAgora.wMinute < 10 THEN
			sAux[3] := CONCAT('0',WORD_TO_STRING(tsAgora.wMinute));
		ELSE
			sAux[3] := WORD_TO_STRING(tsAgora.wMinute);
		END_IF
		sAux[4] := ':';
		
		IF tsAgora.wSecond < 10 THEN
			sAux[5] := CONCAT('0',WORD_TO_STRING(tsAgora.wSecond));
		ELSE
			sAux[5] := WORD_TO_STRING(tsAgora.wSecond);
		END_IF
		sAux2 := F_ConcatArray(sAux);
		
		
		FOR I := iMinVetor TO iMaxVetor DO
			Vetor[I].x :=  sAux2;
		END_FOR
		
	
	END_IF
	
	
	
	tonControle.in := TRUE;
	
	IF tonControle.q THEN
		tonControle.in := FALSE;
		
		FOR I := iMinVetor TO iMaxVetor DO
			Vetor[I].y := Vetor[I+1].y;
			Vetor[I].x := Vetor[I+1].x;
		END_FOR
		
		Vetor[iMaxVetor].y := (Valor);
		
		IF emXColocarTimespamp THEN
			sAux[1] := WORD_TO_STRING(tsAgora.wHour);
			sAux[2] := ':';
			sAux[3] := WORD_TO_STRING(tsAgora.wMinute);
			sAux[4] := ':';
			sAux[5] := WORD_TO_STRING(tsAgora.wSecond);
			Vetor[iMaxVetor].x := F_ConcatArray(sAux);
		ELSE
			FOR I := iMinVetor TO iMaxVetor DO
				Vetor[I].x := '';
			END_FOR
		END_IF
		
		
		
	END_IF
	
	tonControle(IN:= , PT:=TempoEntreCadaAmostra , Q=> , ET=> );


ELSE
	ValidaLicensa();
END_IF

END_FUNCTION_BLOCK

// FBs/TEMPORARIO TROCAR DE BLIBLIOTECA/FB_ControleValvula
FUNCTION_BLOCK FB_ControleValvula
VAR_INPUT
	xAutomaticoManual 	: BOOL;
	xLigaManu			: BOOL;
	xLigaAuto			: BOOL;
	xBloqueio			: BOOL;
	xEmergenciaOK		: BOOL;
	xFeedBackValvula	: BOOL;
	xByPassFeedBack		: BOOL;
	xResetContador		: BOOL;
	rTempoFeedBackSeg	: REAL;
	sNome_Funcao		: STRING;
	xNormalmenteAberto	: BOOL;
END_VAR
VAR_OUTPUT
	xSaidaValvula		: BOOL;
	iStsValvula			: INT;
	iSucessoAionamento	: INT;
	iFalhaAcionamento	: INT;
END_VAR
VAR
	tonFeedBack : TON;
	rtAcionou	: R_TRIG;
	rtFalha		: R_TRIG;
END_VAR


IF xLicensaValida87208720 THEN	
	
	Controle();
	
	Status();

ELSE
	ValidaLicensa();
END_IF

ACTION Controle:





xSaidaValvula := FALSE;


IF xEmergenciaOK AND NOT xBloqueio THEN
	IF xAutomaticoManual THEN
		xSaidaValvula := xLigaAuto;
	ELSE
		xSaidaValvula := xLigaManu;
	END_IF

END_IF


tonFeedBack(IN:=xSaidaValvula AND NOT (xByPassFeedBack OR xFeedBackValvula), PT:=TO_TIME(rTempoFeedBackSeg*1000) , Q=> , ET=> );

(*
IF tonFeedBack.q AND NOT xFeedBackValvula THEN
	xSaidaValvula := FALSE;
END_IF
*)
END_ACTION

ACTION Status:

IF NOT xNormalmenteAberto THEN
	
	iStsValvula := 1;//Fechada em automatico
	
	IF NOT xAutomaticoManual THEN
		iStsValvula := 2;//Fechada em manual
	END_IF
	
	IF xSaidaValvula AND (xFeedBackValvula OR xByPassFeedBack) THEN
		IF xAutomaticoManual THEN
			iStsValvula := 3; // acionada Automatico
		ELSE
			iStsValvula := 4; // acionada Manual
		END_IF
	END_IF
	
	IF xBloqueio THEN
		iStsValvula := 5; // bloqueada
	END_IF
	
	IF tonFeedBack.q THEN
		iStsValvula := 6; // falha // faha feedback
	END_IF
	
	IF NOT xEmergenciaOK THEN
		iStsValvula := 7; // Emergencia
	END_IF
	
	
	rtAcionou(CLK:= iStsValvula = 4 OR iStsValvula = 3, Q=> );
	IF rtAcionou.q THEN
		iSucessoAionamento := iSucessoAionamento +1;
	END_IF
	
	rtFalha(CLK:= iStsValvula = 6, Q=> );
	IF rtFalha.q THEN
		iFalhaAcionamento := iFalhaAcionamento +1;
	END_IF

ELSE
	
	
	
	IF xAutomaticoManual THEN
		iStsValvula := 3;//Fechada em manual
	ELSE
		iStsValvula := 4;//Fechada em automatico
	END_IF
	
	
	IF xSaidaValvula AND (xFeedBackValvula OR xByPassFeedBack) THEN
		IF xAutomaticoManual THEN
			iStsValvula := 1; // acionada Automatico
		ELSE
			iStsValvula := 2; // acionada Manual
		END_IF
	END_IF
	
	
	IF xBloqueio THEN
		iStsValvula := 5; // bloqueada
	END_IF
	
	IF tonFeedBack.q THEN
		iStsValvula := 6; // falha // faha feedback
	END_IF
	
	IF NOT xEmergenciaOK THEN
		iStsValvula := 7; // Emergencia
	END_IF
	
	
	rtAcionou(CLK:= iStsValvula = 4 OR iStsValvula = 3, Q=> );
	IF rtAcionou.q THEN
		iSucessoAionamento := iSucessoAionamento +1;
	END_IF
	
	rtFalha(CLK:= iStsValvula = 6, Q=> );
	IF rtFalha.q THEN
		iFalhaAcionamento := iFalhaAcionamento +1;
	END_IF


END_IF
END_ACTION

END_FUNCTION_BLOCK

// FUNs/TempoParaString/F_TempoEmStringAteHoras
FUNCTION F_TempoEmStringAteHoras : STRING
VAR_INPUT
	Tempo				: TIME;	// tempo a ser transformado em string
	xMostraHoras		: BOOL;	// se mostra horas
	xMostraMinutos		: BOOL;	// se mostra minutos
	xMostraSegundos		: BOOL;	// se mostras segundos
	xMostraMilisegundos	: BOOL;	// se mostra milisegundos
	xCascata			: BOOL;	// se sobrar algum tempo ele joga no proximo que vai ser mostrado
END_VAR
VAR
	sAux	: ARRAY[0..20] OF STRING(255);
	stTempo	: OTSTRUCT;
END_VAR


IF xLicensaValida87208720 THEN	
		
	
	stTempo := TIME_TO_OTSTRUCT(Tempo);
	
	IF xMostraHoras THEN
		IF stTempo.wHour < 10 THEN
			sAux[1]	:= '0';
			sAux[2]	:= TO_STRING(stTempo.wHour);
		ELSE
			sAux[1]	:= '';
			sAux[2]	:= TO_STRING(stTempo.wHour);
		END_IF
	END_IF
	
	IF xMostraMinutos THEN
	
		IF xMostraHoras THEN
			sAux[3] := ':';
		END_IF
	
		IF stTempo.wMinute < 10 THEN
			sAux[4]	:= '0';
			sAux[5]	:= TO_STRING(stTempo.wMinute);
		ELSE
			sAux[4]	:= '';
			sAux[5]	:= TO_STRING(stTempo.wMinute);
		END_IF
	END_IF
	
	IF xMostraSegundos THEN
	
		IF xMostraHoras OR xMostraMinutos THEN
			sAux[6] := ':';
		END_IF
	
		IF stTempo.wSecond < 10 THEN
			sAux[7]	:= '0';
			sAux[8]	:= TO_STRING(stTempo.wSecond);
		ELSE
			sAux[7]	:= '';
			sAux[8]	:= TO_STRING(stTempo.wSecond);
		END_IF
	END_IF
	
	IF xMostraMilisegundos THEN
	
		IF xMostraHoras OR xMostraMinutos OR xMostraSegundos THEN
			sAux[9] := '.';
		END_IF
	
		IF stTempo.wMilliseconds < 10 THEN
			sAux[10]	:= '0';
			sAux[11]	:= TO_STRING(stTempo.wMilliseconds);
		ELSE
			sAux[10]	:= '';
			sAux[11]	:= TO_STRING(stTempo.wMilliseconds);
		END_IF
	END_IF
	
	F_TempoEmStringAteHoras := F_ConcatArray(sAux);
	
ELSE
	F_TempoEmStringAteHoras := '';
END_IF

END_FUNCTION

// FUNs/F_ConcatArray1000
FUNCTION F_ConcatArray1000 : STRING(1000) //Concatena um array de string
VAR_IN_OUT
	sArray : ARRAY[*] OF STRING(80);
END_VAR
VAR
	iTamanhoArray : INT;
	iTamanhoMinArray : INT;
	i : INT;
END_VAR


IF xLicensaValida87208720 THEN	
		
	
	//Criado por Tiago Bortolini Cunico
	
	iTamanhoArray := DINT_TO_INT(UPPER_BOUND(sArray,1));
	iTamanhoMinArray := DINT_TO_INT(LOWER_BOUND(sArray,1));
	
	FOR i := iTamanhoMinArray TO iTamanhoArray DO
		CONCAT2(pSrcString1:= ADR(F_ConcatArray1000), pSrcString2:= ADR(sArray[i]), pDstString:= ADR(F_ConcatArray1000), nDstSize:= SIZEOF(F_ConcatArray1000));
	END_FOR
	
ELSE
	F_ConcatArray1000 := '';
	ValidaLicensa();
END_IF

END_FUNCTION

// FUNs/F_ConcatArray10000
FUNCTION F_ConcatArray10000 : STRING(10000) //Concatena um array de string
VAR_IN_OUT
	sArray : ARRAY[*] OF STRING(80);
END_VAR
VAR
	iTamanhoArray : INT;
	iTamanhoMinArray : INT;
	i : INT;
END_VAR


IF xLicensaValida87208720 THEN	
		
	
	//Criado por Tiago Bortolini Cunico
	
	iTamanhoArray := DINT_TO_INT(UPPER_BOUND(sArray,1));
	iTamanhoMinArray := DINT_TO_INT(LOWER_BOUND(sArray,1));
	
	FOR i := iTamanhoMinArray TO iTamanhoArray DO
		CONCAT2(pSrcString1:= ADR(F_ConcatArray10000), pSrcString2:= ADR(sArray[i]), pDstString:= ADR(F_ConcatArray10000), nDstSize:= SIZEOF(F_ConcatArray10000));
	END_FOR
	
ELSE
	F_ConcatArray10000 := '';
	ValidaLicensa();
END_IF

END_FUNCTION

// FUNs/F_EntradaEmPorcentagem
FUNCTION F_EntradaEmPorcentagem : INT
VAR_INPUT
	Entrada : INT;
	maxi	: INT := 1800;
END_VAR
VAR
END_VAR

IF xLicensaValida87208720 THEN
	
	
	F_EntradaEmPorcentagem := REAL_TO_INT(
								 SCALE_R(
									X:= Entrada, 
									I_LO:= 0, 
									I_HI:= 100, 
									O_LO:= 0, 
									O_HI:= maxi));
ELSE
	F_EntradaEmPorcentagem := 0;	
	ValidaLicensa();						
END_IF

END_FUNCTION

// FUNs/F_EstruturaDiferente
(* 
:Descrição: Função para comparação de estruturas.

:Instruçoes de uso: Passar o endereço para a primeira estrutura, pra segunda e o tamanho dela. Fica tipo assim "xAux := F_EstruturaDiferente(pEstrutura1:=ADR(Teste1), pEstrutura2:=ADR(Teste2), pTamanhoEstrutura:=SIZEOF(ADR(Teste1)));". 

*Cuidado, essa função pode gerar erro de referencia. Principalmente quando muda a estrutura online. Recomendado o uso do check pointer*

*)

{attribute 'hide_all_locals'}
FUNCTION F_EstruturaDiferente : BOOL
VAR_INPUT
	pEstrutura1 : POINTER TO BYTE;
	pEstrutura2 : POINTER TO BYTE;
	pTamanhoEstrutura : UDINT;
END_VAR
VAR
	i: UDINT;
	bEstrutura1 : BYTE;
	bEstrutura2 : BYTE;
	pAux : POINTER TO BYTE;
END_VAR

IF xLicensaValida87208720 THEN
	FOR i:= 0 TO pTamanhoEstrutura DO
		pAux := (pEstrutura1+i);
		bEstrutura1 := pAux^;
		
		pAux := (pEstrutura2+i);
		bEstrutura2 := pAux^;
		
		F_EstruturaDiferente := F_EstruturaDiferente OR (bEstrutura1 <> bEstrutura2);
	END_FOR
	F_EstruturaDiferente := FALSE;
ELSE
	ValidaLicensa();
END_IF

END_FUNCTION

// FUNs/F_LimpaArrayString
FUNCTION F_LimpaArrayString : string(255) //Concatena um array de string
VAR_IN_OUT
	sArray : ARRAY[*] OF STRING(255);
END_VAR
VAR
	iTamanhoArray : INT;
	iTamanhoMinArray : INT;
	i : INT;
END_VAR

IF xLicensaValida87208720 THEN
	//Criado por Tiago Bortolini Cunico
	
	iTamanhoArray := DINT_TO_INT(UPPER_BOUND(sArray,1));
	iTamanhoMinArray := DINT_TO_INT(LOWER_BOUND(sArray,1));
	
	FOR i := iTamanhoMinArray TO iTamanhoArray DO
		sArray[i] := '';
	END_FOR

ELSE
	ValidaLicensa();
	F_LimpaArrayString := '';
END_IF

END_FUNCTION

// FUNs/F_LimpaDataBase
FUNCTION F_LimpaDataBase : BOOL
VAR_IN_OUT
	DataBase : ARRAY[*,*] OF STRING(255);
END_VAR
VAR
	i,j : DINT := 0;
END_VAR

IF xLicensaValida87208720 THEN

	FOR i:= LOWER_BOUND(DataBase,1) TO UPPER_BOUND(DataBase,1) DO
		FOR j:= LOWER_BOUND(DataBase,2) TO UPPER_BOUND(DataBase,2) DO
			DataBase[i,j] := '';
		END_FOR
	END_FOR
	
	
	F_LimpaDataBase := TRUE;
ELSE
	ValidaLicensa();
	F_LimpaDataBase := FALSE;
END_IF

END_FUNCTION

// FUNs/F_MaisOuMenos
FUNCTION F_MaisOuMenos : BOOL// descrição 1
// descrição 2
VAR_INPUT
	Valor : ANY_NUM;
	Comparado : ANY_NUM;
	PorcentAcima : REAL;
	PorcentAbaixo : REAL;
END_VAR
VAR
	rValor : REAL;
	rComparado : REAL;
	rPorcentAcima : REAL;
	rPorcentAbaixo : REAL;
	abaixo : REAL;
	acima : REAL;
	pRealAux : POINTER TO REAL;
	pIntAux : POINTER TO INT;
END_VAR

IF xLicensaValida87208720 THEN

	
	IF (Valor.TypeClass = __SYSTEM.TYPE_CLASS.TYPE_REAL) THEN
		pRealAux := Valor.pValue;
		rValor := ABS(pRealAux^);
	ELSE
		pIntAux := Valor.pValue;
		rValor := ABS(INT_TO_REAL(pIntAux^));
	END_IF
	
	
	IF (Comparado.TypeClass = __SYSTEM.TYPE_CLASS.TYPE_REAL) THEN
		pRealAux := Comparado.pValue;
		rComparado := ABS(pRealAux^);
	ELSE
		pIntAux := Comparado.pValue;
		rComparado := ABS(INT_TO_REAL(pIntAux^));
	END_IF
	
	
	//rComparado := TO_REAL(Comparado.pValue^);
	rPorcentAcima := PorcentAcima;//TO_REAL(PorcentAcima.pValue^);
	rPorcentAbaixo := PorcentAbaixo; //TO_REAL(PorcentAbaixo.pValue^);
	
	abaixo := rComparado*(1-rPorcentAbaixo/100);
	acima := rComparado*(1+rPorcentAcima/100);
	
	F_MaisOuMenos := abaixo<=rValor AND rValor<=acima;
	
ELSE
	ValidaLicensa();
	F_MaisOuMenos := FALSE;
END_IF

END_FUNCTION

// FUNs/F_RetiraCasa
FUNCTION F_RetiraCasa : REAL
VAR_INPUT
	Entrada : REAL;
	casa : INT;
END_VAR
VAR
	rAux : REAL;
END_VAR

IF xLicensaValida87208720 THEN

	rAux := DINT_TO_REAL(TRUNC(Entrada*(casa*10)));
	F_RetiraCasa := rAux/(casa*10);

ELSE
	ValidaLicensa();
	F_RetiraCasa := 0;
END_IF

END_FUNCTION

// FUNs/F_StringSeparadorArrayInt
FUNCTION F_StringSeparadorArrayInt : BOOL
VAR_INPUT
	sStr : STRING;
	sSeparador : STRING;
END_VAR
VAR_IN_OUT
	ListaINT : ARRAY[*] OF INT;
END_VAR
VAR
	iListIntMIN : INT;
	iListIntMAX : INT;
	
	sParteEsquerda : STRING;
	sResto : STRING;
	sSepara : STRING;
	
	iIndex : INT;
END_VAR


iListIntMIN := DINT_TO_INT(LOWER_BOUND(ListaINT,1));
iListIntMAX := DINT_TO_INT(UPPER_BOUND(ListaINT,1));


sSepara := sStr;
iIndex := iListIntMIN;

WHILE FindAndSplit(
		pSeparator:= ADR(sSeparador), 
		pSrcString:= ADR(sSepara), 
		pLeftString:= ADR(sParteEsquerda), 
		nLeftSize:= SIZEOF(sParteEsquerda), 
		pRightString:= ADR(sResto), 
		nRightSize:= SIZEOF(sResto), 
		bSearchFromRight:= FALSE) DO
	
	
	ListaINT[iIndex]:= STRING_TO_INT(sParteEsquerda);	
	sSepara := sResto;
	
	iIndex := iIndex + 1;
	
	IF iIndex > iListIntMAX THEN
		F_StringSeparadorArrayInt := FALSE;
		EXIT;
	END_IF
	
END_WHILE

F_StringSeparadorArrayInt := TRUE;

END_FUNCTION

// FUNs/F_StringSeparadorArrayInt_1
FUNCTION F_StringSeparadorArrayInt_1 : BOOL
VAR_INPUT
	sStr : STRING;
	sSeparador : STRING;
END_VAR
VAR_IN_OUT
	ListaINT : ARRAY[*] OF INT;
END_VAR
VAR
	iListIntMIN : INT;
	iListIntMAX : INT;
	
	sParteEsquerda : STRING;
	sResto : STRING;
	sSepara : STRING;
	
	iIndex : INT;
END_VAR


iListIntMIN := DINT_TO_INT(LOWER_BOUND(ListaINT,1));
iListIntMAX := DINT_TO_INT(UPPER_BOUND(ListaINT,1));


sSepara := sStr;
iIndex := iListIntMIN;

WHILE FindAndSplit(
		pSeparator:= ADR(sSeparador), 
		pSrcString:= ADR(sSepara), 
		pLeftString:= ADR(sParteEsquerda), 
		nLeftSize:= SIZEOF(sParteEsquerda), 
		pRightString:= ADR(sResto), 
		nRightSize:= SIZEOF(sResto), 
		bSearchFromRight:= FALSE) DO
	
	
	ListaINT[iIndex]:= STRING_TO_INT(sParteEsquerda);	
	sSepara := sResto;
	
	iIndex := iIndex + 1;
	
	IF iIndex > iListIntMAX THEN
		F_StringSeparadorArrayInt := FALSE;
		EXIT;
	END_IF
	
END_WHILE

F_StringSeparadorArrayInt := TRUE;

END_FUNCTION

// POUs/Main
PROGRAM Main
VAR

	r1 : REAL;
	r2 : REAL;
	xAux : BOOL;


END_VAR





xAux := F_MaisOuMenos(Valor:= r1, Comparado:= r2, PorcentAcima:= 5, PorcentAbaixo:= 5);

END_PROGRAM

// Project Information/F_GetCompany
// This function has been automatically generated from the project information.
{attribute 'signature_flag' := '1073741824'}
{attribute 'TcGenerated'}
{attribute 'no-analysis'}
FUNCTION F_GetCompany : WSTRING
VAR_INPUT
	
END_VAR

F_GetCompany := "Teknike";

END_FUNCTION

// Project Information/F_GetTitle
// This function has been automatically generated from the project information.
{attribute 'signature_flag' := '1073741824'}
{attribute 'TcGenerated'}
{attribute 'no-analysis'}
FUNCTION F_GetTitle : WSTRING
VAR_INPUT
	
END_VAR

F_GetTitle := "Geral";

END_FUNCTION

// Project Information/F_GetVersion
// This function has been automatically generated from the project information.
{attribute 'signature_flag' := '1073741824'}
{attribute 'TcGenerated'}
{attribute 'no-analysis'}
FUNCTION F_GetVersion : ST_LibVersion
VAR_INPUT
	
END_VAR

F_GetVersion.iMajor := 2;
F_GetVersion.iMinor := 0;
F_GetVersion.iBuild := 16;
F_GetVersion.iRevision := 0;
F_GetVersion.sVersion := '2.0.16';
F_GetVersion.nFlags := 0;

END_FUNCTION
